Yaskawa INFORM job: N_R2_D7,1(-165,-90)0.JBI

/JOB
//NAME N_R2_D7,1(-165,-90)0
//POS
///NPOS 215,215,215,10,0,0
///TOOL 0
///POSTYPE PULSE
///PULSE
C00000=-39723,-76225,-106677,19950,71807,76871
C00001=-136716,-73683,-105524,19345,72156,77265
C00002=-161407,-91524,-110310,15012,103390,71507
C00003=-134262,-92612,-59078,787,74622,77224
C00004=-134610,-92069,-54626,808,72165,77088
C00005=-134755,-91759,-52790,817,71196,77032
C00006=-134778,-90628,-50545,822,70395,77019
C00007=-134779,-90815,-50888,821,70510,77019
C00008=-134780,-90766,-50877,821,70529,77019
C00009=-135151,-92885,-51740,837,69975,76888
C00010=-134780,-90766,-50877,821,70529,77019
C00011=-134635,-91110,-52736,812,71495,77075
C00012=-134286,-91743,-57244,790,73940,77211
C00013=-131535,-88408,-77632,452,88335,78233
C00014=-134472,-105055,-82285,1702,77673,77142
C00015=-134729,-104914,-78076,1744,75161,77018
C00016=-134834,-104745,-76339,1762,74182,76968
C00017=-134858,-103911,-74317,1771,73367,76948
C00018=-134859,-104062,-74637,1770,73487,76949
C00019=-134909,-103988,-74547,1775,73470,76931
C00020=-135283,-106552,-75509,1819,72754,76790
C00021=-134909,-103988,-74547,1775,73470,76931
C00022=-134803,-104200,-76305,1757,74440,76982
C00023=-134544,-104461,-80571,1713,76925,77107
C00024=-136082,-134381,-102209,6463,55903,75707
C00025=-135108,-114579,-94528,5981,61099,76375
C00026=-134953,-111416,-89269,6014,59485,76347
C00027=-134891,-110125,-87144,6029,58840,76336
C00028=-134915,-109472,-85222,6092,57999,76280
C00029=-134915,-109614,-85578,6083,58144,76288
C00030=-134962,-109452,-85494,6099,58179,76271
C00031=-135337,-112331,-86541,6305,57378,76076
C00032=-134962,-109452,-85494,6099,58179,76271
C00033=-135023,-110765,-87631,6083,58821,76283
C00034=-135179,-113988,-92923,6048,60424,76311
C00035=-156260,-82084,-105549,20460,72443,69801
C00036=-137260,-84248,-120477,10166,77039,76481
C00037=-137260,-138866,-129024,10166,31486,76481
C00038=-31464,-162597,-129024,10166,12061,76481
C00039=11401,-148032,-125424,11666,35639,75770
C00040=126224,-114648,-117374,36487,17100,65054
C00041=160935,-140982,-109639,13467,75088,4607
C00042=171546,-94218,-58921,11830,67408,-77190
C00043=173316,-92720,-54117,11803,65014,-76792
C00044=174042,-92038,-52145,11792,64066,-76624
C00045=174183,-90834,-49869,11851,63281,-76655
C00046=174042,-92038,-52145,11792,64066,-76624
C00047=174177,-91005,-50226,11839,63410,-76643
C00048=175494,-92657,-50922,11711,62814,-76221
C00049=174177,-91005,-50226,11839,63410,-76643
C00050=173449,-91716,-52219,11847,64356,-76811
C00051=171674,-93290,-57074,11869,66744,-77212
C00052=148466,-121612,-87036,17170,72641,-74850
C00053=158367,-105008,-80303,12719,76823,-80933
C00054=159865,-104818,-76175,12706,74203,-80677
C00055=160482,-104628,-74471,12705,73177,-80565
C00056=160593,-103709,-72411,12744,72384,-80610
C00057=160482,-104628,-74471,12705,73177,-80565
C00058=160542,-103788,-72707,12740,72530,-80613
C00059=161564,-106010,-73554,12683,71765,-80329
C00060=160542,-103788,-72707,12740,72530,-80613
C00061=159923,-104017,-74432,12740,73548,-80725
C00062=158422,-104310,-78610,12746,76147,-80984
C00063=158674,-141756,-113025,9949,80411,-74851
C00064=158893,-111477,-96824,9930,85641,-81694
C00065=159967,-112919,-93343,9895,82666,-81559
C00066=160412,-113323,-91879,9887,81519,-81496
C00067=160523,-112689,-89977,9898,80673,-81526
C00068=160509,-112801,-90280,9896,80802,-81520
C00069=160550,-112812,-90284,9894,80794,-81506
C00070=161574,-115499,-91253,9843,79895,-81223
C00071=160550,-112812,-90284,9894,80794,-81506
C00072=160103,-112470,-91772,9900,81925,-81571
C00073=159023,-111201,-95321,9929,84853,-81711
C00074=160752,-88554,-104051,4755,98097,-77411
C00075=135358,-109973,-92009,-1179,81206,-77087
C00076=132931,-92872,-58798,-293,74315,-77659
C00077=133296,-92294,-54326,-308,71862,-77528
C00078=133447,-91972,-52482,-315,70894,-77474
C00079=133488,-90828,-50231,-318,70096,-77458
C00080=133482,-91042,-50637,-317,70236,-77460
C00081=133460,-91107,-50617,-317,70190,-77467
C00082=133801,-93226,-51476,-330,69631,-77349
C00083=133460,-91107,-50617,-317,70190,-77467
C00084=133307,-91465,-52485,-310,71155,-77522
C00085=132941,-92137,-57014,-294,73596,-77654
C00086=138453,-137227,-94273,-1895,68830,-75577
C00087=132988,-105621,-81970,-1125,77172,-77601
C00088=133268,-105409,-77729,-1165,74675,-77481
C00089=133383,-105214,-75980,-1182,73700,-77431
C00090=133423,-104355,-73948,-1190,72892,-77409
C00091=133417,-104520,-74315,-1189,73033,-77413
C00092=133393,-104538,-74287,-1187,73006,-77421
C00093=133734,-107100,-75243,-1226,72284,-77295
C00094=133393,-104538,-74287,-1187,73006,-77421
C00095=133278,-104776,-76057,-1170,73972,-77470
C00096=132997,-105102,-80353,-1129,76444,-77591
C00097=138253,-142244,-101762,-7760,51895,-74453
C00098=133458,-115366,-94293,-4986,60456,-76916
C00099=133364,-112113,-89005,-5028,58873,-76880
C00100=133327,-110790,-86870,-5046,58239,-76865
C00101=133368,-110104,-84936,-5108,57407,-76810
C00102=133362,-110233,-85266,-5098,57543,-76819
C00103=133377,-110217,-85238,-5104,57535,-76813
C00104=133717,-113094,-86276,-5290,56721,-76638
C00105=133377,-110217,-85238,-5104,57535,-76813
C00106=133414,-111565,-87387,-5085,58165,-76828
C00107=133508,-114885,-92709,-5041,59734,-76864
C00108=141804,-106560,-89724,-13944,62113,-73509
C00109=139379,-94179,-83096,-11060,68876,-75147
C00110=139056,-93239,-80222,-11055,67569,-75143
C00111=138655,-90526,-79037,-10882,68167,-75347
C00112=139020,-93447,-81559,-10991,68267,-75222
C00113=135650,-94437,-80689,-10014,66800,-76334
C00114=131133,-95634,-81147,-8583,65949,-77941
C00115=127606,-96266,-81385,-7430,65422,-79216
C00116=127923,-97381,-84321,-7467,66675,-79179
C00117=129037,-107781,-90700,-8626,61514,-78396
C00118=153259,-105355,-101722,-11659,72368,-68227
C00119=139055,-107982,-91136,13627,98522,-80003
C00120=140531,-111621,-88895,13695,95112,-79863
C00121=141160,-112889,-87907,13741,93781,-79791
C00122=141114,-113409,-89355,13751,94395,-79738
C00123=140635,-110012,-86860,13696,94681,-79874
C00124=145054,-111200,-87361,14229,93626,-78446
C00125=149927,-108602,-86499,14790,93534,-76747
C00126=153516,-106318,-85721,15167,93544,-75484
C00127=152717,-105120,-86692,15125,94866,-75603
C00128=150826,-101669,-88898,15064,98245,-75855
C00129=161013,-93310,-79433,24228,97681,-73156
C00130=152044,-102420,-74574,18748,88667,-80737
C00131=154129,-104098,-71555,18965,85609,-80472
C00132=155013,-104629,-70277,19068,84402,-80349
C00133=154938,-105384,-71853,19049,84971,-80287
C00134=154138,-102381,-69420,18973,85198,-80533
C00135=158674,-102440,-69551,19374,84196,-79089
C00136=163166,-99303,-68473,19685,84034,-77522
C00137=166415,-96688,-67542,19865,83984,-76373
C00138=165435,-96203,-68797,19786,85183,-76526
C00139=163100,-94647,-71761,19624,88219,-76868
C00140=177469,-96162,-81466,-5174,90371,-76160
C00141=140989,-97571,-77910,-6477,80304,-75413
C00142=139257,-88771,-70558,-5122,84704,-76235
C00143=139247,-89361,-68393,-5133,83074,-76172
C00144=138839,-86919,-67301,-5121,83628,-76333
C00145=139210,-89792,-69844,-5127,83741,-76212
C00146=135828,-90440,-68818,-5070,82565,-77317
C00147=131175,-91540,-69244,-4968,81974,-78881
C00148=127631,-92103,-69459,-4877,81601,-80076
C00149=127824,-91599,-71673,-4868,83228,-80074
C00150=128905,-101797,-79416,-5532,77763,-79457
C00151=137935,-111344,-72360,-1825,88711,-76983
C00152=138175,-87355,-54576,-1641,89871,-76939
C00153=138462,-88899,-51460,-1591,87166,-76810
C00154=138585,-89409,-50143,-1570,86097,-76756
C00155=138142,-87310,-49251,-1647,86617,-76908
C00156=138544,-90243,-51824,-1577,86701,-76777
C00157=134711,-90264,-50450,-2245,85757,-78018
C00158=129567,-91064,-50732,-3132,85354,-79692
C00159=133440,-90680,-49995,-7180,85761,-79174
C00160=133642,-90171,-51309,-7139,86839,-79169
C00161=134115,-88628,-54418,-7054,89566,-79166
C00162=164381,-109390,-67526,9871,79554,-67793
C00163=178481,-110687,-72352,20846,77564,-61880
C00164=158703,-97120,-53511,19723,77491,-80168
C00165=161312,-97088,-49613,20147,74642,-79736
C00166=162421,-96967,-47993,20332,73505,-79545
C00167=162322,-98010,-49764,20272,74049,-79485
C00168=161267,-95191,-47313,20182,74238,-79821
C00169=166229,-94856,-47327,20585,73246,-78256
C00170=170826,-91864,-46338,20811,73023,-76672
C00171=170725,-92212,-45770,23236,70848,-76635
C00172=169440,-92471,-47412,23069,72000,-76869
C00173=166376,-92848,-51371,22679,74886,-77407
C00174=149893,-144723,-110594,14593,75698,-63607
C00175=126224,-114648,-117374,36487,17100,65054
C00176=118781,-153852,-129024,32591,23356,65054
C00177=12469,-167082,-125424,11666,16324,75770
C00178=-137258,-84249,-120477,10166,64820,76481
C00179=-160540,-100856,-113062,23154,68828,67580
C00180=-142919,-103613,-89511,14221,64514,73447
C00181=-140713,-93202,-83145,11806,69584,74803
C00182=-140366,-92325,-80297,11799,68258,74797
C00183=-140342,-92507,-81623,11736,68962,74877
C00184=-139943,-89620,-79106,11620,68840,75011
C00185=-137000,-93615,-80822,10786,67454,75962
C00186=-132529,-94936,-81358,9390,66550,77539
C00187=-129034,-95667,-81655,8259,65976,78791
C00188=-129377,-96731,-84569,8298,67246,78755
C00189=-130985,-110873,-91431,10312,58832,77470
C00190=-137786,-122665,-93672,6634,76519,76374
C00191=-142705,-98537,-78672,7318,79679,74834
C00192=-140492,-88091,-70749,5581,85268,75891
C00193=-140474,-88727,-68610,5592,83630,75824
C00194=-140449,-89137,-70051,5586,84302,75862
C00195=-140046,-86288,-67512,5580,84176,75994
C00196=-137092,-89887,-69090,5534,83097,76954
C00197=-132483,-91099,-69589,5437,82469,78500
C00198=-128968,-91749,-69858,5349,82066,79683
C00199=-129166,-91202,-72049,5340,83701,79685
C00200=-130908,-106571,-81390,6599,74332,78625
C00201=-147199,-111997,-78117,4842,93237,75003
C00202=-140629,-86347,-53809,6324,90898,77078
C00203=-140437,-88027,-50796,6352,88182,77004
C00204=-140355,-88591,-49520,6369,87107,76977
C00205=-140327,-89422,-51202,6373,87709,77017
C00206=-139876,-86509,-48628,6458,87588,77159
C00207=-136525,-89545,-49887,7080,86535,78207
C00208=-131427,-90479,-50246,8002,85818,79842
C00209=-127439,-90954,-50432,8701,85292,81122
C00210=-127780,-90460,-51749,8636,86380,81084
C00211=-128575,-88953,-54867,8495,89126,81007
C00212=-161407,-91524,-110310,15012,103390,71507
C00213=-136716,-73683,-105524,19345,72156,77265
C00214=-39723,-76225,-106677,19950,71807,76871
BC00000=295325,674563,1075175
BC00001=353535,895977,1075175
BC00002=353535,975867,1075175
BC00003=346138,1016365,1074941
BC00004=346138,1016365,1074941
BC00005=346138,1016365,1074941
BC00006=346138,1016365,1074941
BC00007=346138,1016365,1074941
BC00008=346138,1016365,1074941
BC00009=346138,1016365,1074941
BC00010=346138,1016365,1074941
BC00011=346138,1016365,1074941
BC00012=346138,1016365,1074941
BC00013=345633,1015596,1047596
BC00014=345436,1039539,1075175
BC00015=345436,1039539,1075175
BC00016=345436,1039539,1075175
BC00017=345436,1039539,1075175
BC00018=345436,1039539,1075175
BC00019=345436,1039539,1075175
BC00020=345436,1039539,1075175
BC00021=345436,1039539,1075175
BC00022=345436,1039539,1075175
BC00023=345436,1039539,1075175
BC00024=345633,1030850,1075175
BC00025=346084,1031619,1075175
BC00026=346084,1031619,1075175
BC00027=346084,1031619,1075175
BC00028=346084,1031619,1075175
BC00029=346084,1031619,1075175
BC00030=346084,1031619,1075175
BC00031=346084,1031619,1075175
BC00032=346084,1031619,1075175
BC00033=346084,1031619,1075175
BC00034=346084,1031619,1075175
BC00035=381896,966588,1075175
BC00036=353816,923989,1075175
BC00037=353816,923989,1075175
BC00038=379773,1126391,1075175
BC00039=398190,1030285,1075175
BC00040=312632,1138057,1075175
BC00041=340753,1115300,1075175
BC00042=317618,1085268,1067802
BC00043=317618,1085268,1067802
BC00044=317618,1085268,1067802
BC00045=317618,1085268,1067802
BC00046=317618,1085268,1067802
BC00047=317618,1085268,1067802
BC00048=317618,1085268,1067802
BC00049=317618,1085268,1067802
BC00050=317618,1085268,1067802
BC00051=317618,1085268,1067802
BC00052=304558,1071386,1075175
BC00053=304527,1061353,1075175
BC00054=304527,1061353,1075175
BC00055=304527,1061353,1075175
BC00056=304527,1061353,1075175
BC00057=304527,1061353,1075175
BC00058=304527,1061353,1075175
BC00059=304527,1061353,1075175
BC00060=304527,1061353,1075175
BC00061=304527,1061353,1075175
BC00062=304527,1061353,1075175
BC00063=297809,1030861,1075175
BC00064=297809,1030861,1075175
BC00065=297809,1030861,1075175
BC00066=297809,1030861,1075175
BC00067=297809,1030861,1075175
BC00068=297809,1030861,1075175
BC00069=297809,1030861,1075175
BC00070=297809,1030861,1075175
BC00071=297809,1030861,1075175
BC00072=297809,1030861,1075175
BC00073=297809,1030861,1075175
BC00074=323405,1100688,1075175
BC00075=345633,1145987,1075175
BC00076=345627,1107551,1074273
BC00077=345627,1107551,1074273
BC00078=345627,1107551,1074273
BC00079=345627,1107551,1074273
BC00080=345627,1107551,1074273
BC00081=345627,1107551,1074273
BC00082=345627,1107551,1074273
BC00083=345627,1107551,1074273
BC00084=345627,1107551,1074273
BC00085=345627,1107551,1074273
BC00086=345633,1085057,1075175
BC00087=345596,1084288,1075175
BC00088=345596,1084288,1075175
BC00089=345596,1084288,1075175
BC00090=345596,1084288,1075175
BC00091=345596,1084288,1075175
BC00092=345596,1084288,1075175
BC00093=345596,1084288,1075175
BC00094=345596,1084288,1075175
BC00095=345596,1084288,1075175
BC00096=345596,1084288,1075175
BC00097=345633,1092894,1075175
BC00098=345573,1092125,1075175
BC00099=345573,1092125,1075175
BC00100=345573,1092125,1075175
BC00101=345573,1092125,1075175
BC00102=345573,1092125,1075175
BC00103=345573,1092125,1075175
BC00104=345573,1092125,1075175
BC00105=345573,1092125,1075175
BC00106=345573,1092125,1075175
BC00107=345573,1092125,1075175
BC00108=338421,1101651,1075175
BC00109=338421,1101651,1075175
BC00110=338421,1101651,1075175
BC00111=338421,1101651,1075175
BC00112=338421,1101651,1075175
BC00113=338421,1101651,1075175
BC00114=338421,1101651,1075175
BC00115=338421,1101651,1075175
BC00116=338421,1101651,1075175
BC00117=338421,1101651,1075175
BC00118=329561,1092894,1075175
BC00119=285121,1016140,1075175
BC00120=285121,1016140,1075175
BC00121=285121,1016140,1075175
BC00122=285121,1016140,1075175
BC00123=285121,1016140,1075175
BC00124=285121,1016140,1075175
BC00125=285121,1016140,1075175
BC00126=285121,1016140,1075175
BC00127=285121,1016140,1075175
BC00128=285121,1016140,1075175
BC00129=322883,1030260,1075175
BC00130=305317,1037338,1075175
BC00131=305317,1037338,1075175
BC00132=305317,1037338,1075175
BC00133=305317,1037338,1075175
BC00134=305317,1037338,1075175
BC00135=305317,1037338,1075175
BC00136=305317,1037338,1075175
BC00137=305317,1037338,1075175
BC00138=305317,1037338,1075175
BC00139=305317,1037338,1075175
BC00140=352461,1065435,1075175
BC00141=338520,1089250,1075175
BC00142=338520,1089250,1075175
BC00143=338520,1089250,1075175
BC00144=338520,1089250,1075175
BC00145=338520,1089250,1075175
BC00146=338520,1089250,1075175
BC00147=338520,1089250,1075175
BC00148=338520,1089250,1075175
BC00149=338520,1089250,1075175
BC00150=338520,1089250,1075175
BC00151=329561,1063988,1075175
BC00152=334879,1082600,1057410
BC00153=334879,1082600,1057410
BC00154=334879,1082600,1057410
BC00155=334879,1082600,1057410
BC00156=334879,1082600,1057410
BC00157=334879,1082600,1057410
BC00158=334879,1082600,1057410
BC00159=334879,1082600,1057410
BC00160=334879,1082600,1057410
BC00161=334879,1082600,1057410
BC00162=331300,1058024,1069499
BC00163=329561,1042367,1075175
BC00164=308437,1059196,1075175
BC00165=308437,1059196,1075175
BC00166=308437,1059196,1075175
BC00167=308437,1059196,1075175
BC00168=308437,1059196,1075175
BC00169=308437,1059196,1075175
BC00170=308437,1059196,1075175
BC00171=308437,1059196,1075175
BC00172=308437,1059196,1075175
BC00173=308437,1059196,1075175
BC00174=340753,1115300,1075175
BC00175=312632,1138057,1075175
BC00176=312632,1138057,1075175
BC00177=398190,1030285,1075175
BC00178=353817,923990,1075175
BC00179=381896,966588,1075175
BC00180=338906,1022094,1075175
BC00181=338906,1022094,1075175
BC00182=338906,1022094,1075175
BC00183=338906,1022094,1075175
BC00184=338906,1022094,1075175
BC00185=338906,1022094,1075175
BC00186=338906,1022094,1075175
BC00187=338906,1022094,1075175
BC00188=338906,1022094,1075175
BC00189=338906,1022094,1075175
BC00190=330026,1050278,1075175
BC00191=338884,1034595,1075175
BC00192=338884,1034595,1075175
BC00193=338884,1034595,1075175
BC00194=338884,1034595,1075175
BC00195=338884,1034595,1075175
BC00196=338884,1034595,1075175
BC00197=338884,1034595,1075175
BC00198=338884,1034595,1075175
BC00199=338884,1034595,1075175
BC00200=338884,1034595,1075175
BC00201=330026,1059203,1075175
BC00202=326517,1040873,1058771
BC00203=326517,1040873,1058771
BC00204=326517,1040873,1058771
BC00205=326517,1040873,1058771
BC00206=326517,1040873,1058771
BC00207=326517,1040873,1058771
BC00208=326517,1040873,1058771
BC00209=326517,1040873,1058771
BC00210=326517,1040873,1058771
BC00211=326517,1040873,1058771
BC00212=353535,975867,1075175
BC00213=353535,895977,1075175
BC00214=295325,674563,1075175
EC00000=-1463287,-556475
EC00001=-1463287,-556475
EC00002=-1463287,-556475
EC00003=-1463287,-556475
EC00004=-1463287,-556475
EC00005=-1463287,-556475
EC00006=-1463287,-556475
EC00007=-1463287,-556475
EC00008=-1463287,-556475
EC00009=-1463287,-556475
EC00010=-1463287,-556475
EC00011=-1463287,-556475
EC00012=-1463287,-556475
EC00013=-1463287,-556475
EC00014=-1463287,-556475
EC00015=-1463287,-556475
EC00016=-1463287,-556475
EC00017=-1463287,-556475
EC00018=-1463287,-556475
EC00019=-1463287,-556475
EC00020=-1463287,-556475
EC00021=-1463287,-556475
EC00022=-1463287,-556475
EC00023=-1463287,-556475
EC00024=-1463287,-556475
EC00025=-1463287,-556475
EC00026=-1463287,-556475
EC00027=-1463287,-556475
EC00028=-1463287,-556475
EC00029=-1463287,-556475
EC00030=-1463287,-556475
EC00031=-1463287,-556475
EC00032=-1463287,-556475
EC00033=-1463287,-556475
EC00034=-1463287,-556475
EC00035=-1463287,-556475
EC00036=-1463287,-556475
EC00037=-1463287,-556475
EC00038=-1463287,-556475
EC00039=-1595090,-3837
EC00040=-1729339,556475
EC00041=-1729339,556475
EC00042=-1729339,556475
EC00043=-1729339,556475
EC00044=-1729339,556475
EC00045=-1729339,556475
EC00046=-1729339,556475
EC00047=-1729339,556475
EC00048=-1729339,556475
EC00049=-1729339,556475
EC00050=-1729339,556475
EC00051=-1729339,556475
EC00052=-1729339,556475
EC00053=-1729339,556475
EC00054=-1729339,556475
EC00055=-1729339,556475
EC00056=-1729339,556475
EC00057=-1729339,556475
EC00058=-1729339,556475
EC00059=-1729339,556475
EC00060=-1729339,556475
EC00061=-1729339,556475
EC00062=-1729339,556475
EC00063=-1729339,556475
EC00064=-1729339,556475
EC00065=-1729339,556475
EC00066=-1729339,556475
EC00067=-1729339,556475
EC00068=-1729339,556475
EC00069=-1729339,556475
EC00070=-1729339,556475
EC00071=-1729339,556475
EC00072=-1729339,556475
EC00073=-1729339,556475
EC00074=-1729339,556475
EC00075=-1729339,556475
EC00076=-1729339,556475
EC00077=-1729339,556475
EC00078=-1729339,556475
EC00079=-1729339,556475
EC00080=-1729339,556475
EC00081=-1729339,556475
EC00082=-1729339,556475
EC00083=-1729339,556475
EC00084=-1729339,556475
EC00085=-1729339,556475
EC00086=-1729339,556475
EC00087=-1729339,556475
EC00088=-1729339,556475
EC00089=-1729339,556475
EC00090=-1729339,556475
EC00091=-1729339,556475
EC00092=-1729339,556475
EC00093=-1729339,556475
EC00094=-1729339,556475
EC00095=-1729339,556475
EC00096=-1729339,556475
EC00097=-1729339,556475
EC00098=-1729339,556475
EC00099=-1729339,556475
EC00100=-1729339,556475
EC00101=-1729339,556475
EC00102=-1729339,556475
EC00103=-1729339,556475
EC00104=-1729339,556475
EC00105=-1729339,556475
EC00106=-1729339,556475
EC00107=-1729339,556475
EC00108=-1729339,556475
EC00109=-1729339,556475
EC00110=-1729339,556475
EC00111=-1729339,556475
EC00112=-1729339,556475
EC00113=-1729339,556475
EC00114=-1729339,556475
EC00115=-1729339,556475
EC00116=-1729339,556475
EC00117=-1729339,556475
EC00118=-1729339,556475
EC00119=-1729339,556475
EC00120=-1729339,556475
EC00121=-1729339,556475
EC00122=-1729339,556475
EC00123=-1729339,556475
EC00124=-1729339,556475
EC00125=-1729339,556475
EC00126=-1729339,556475
EC00127=-1729339,556475
EC00128=-1729339,556475
EC00129=-1729339,556475
EC00130=-1729339,556475
EC00131=-1729339,556475
EC00132=-1729339,556475
EC00133=-1729339,556475
EC00134=-1729339,556475
EC00135=-1729339,556475
EC00136=-1729339,556475
EC00137=-1729339,556475
EC00138=-1729339,556475
EC00139=-1729339,556475
EC00140=-1729339,556475
EC00141=-1729339,556475
EC00142=-1729339,556475
EC00143=-1729339,556475
EC00144=-1729339,556475
EC00145=-1729339,556475
EC00146=-1729339,556475
EC00147=-1729339,556475
EC00148=-1729339,556475
EC00149=-1729339,556475
EC00150=-1729339,556475
EC00151=-1729339,556475
EC00152=-1729339,556475
EC00153=-1729339,556475
EC00154=-1729339,556475
EC00155=-1729339,556475
EC00156=-1729339,556475
EC00157=-1729339,556475
EC00158=-1729339,556475
EC00159=-1729339,556475
EC00160=-1729339,556475
EC00161=-1729339,556475
EC00162=-1729339,556475
EC00163=-1729339,556475
EC00164=-1729339,556475
EC00165=-1729339,556475
EC00166=-1729339,556475
EC00167=-1729339,556475
EC00168=-1729339,556475
EC00169=-1729339,556475
EC00170=-1729339,556475
EC00171=-1729339,556475
EC00172=-1729339,556475
EC00173=-1729339,556475
EC00174=-1729339,556475
EC00175=-1729339,556475
EC00176=-1729339,556475
EC00177=-1595090,-3837
EC00178=-1463287,-556475
EC00179=-1463287,-556475
EC00180=-1463287,-556475
EC00181=-1463287,-556475
EC00182=-1463287,-556475
EC00183=-1463287,-556475
EC00184=-1463287,-556475
EC00185=-1463287,-556475
EC00186=-1463287,-556475
EC00187=-1463287,-556475
EC00188=-1463287,-556475
EC00189=-1463287,-556475
EC00190=-1463287,-556475
EC00191=-1463287,-556475
EC00192=-1463287,-556475
EC00193=-1463287,-556475
EC00194=-1463287,-556475
EC00195=-1463287,-556475
EC00196=-1463287,-556475
EC00197=-1463287,-556475
EC00198=-1463287,-556475
EC00199=-1463287,-556475
EC00200=-1463287,-556475
EC00201=-1463287,-556475
EC00202=-1463287,-556475
EC00203=-1463287,-556475
EC00204=-1463287,-556475
EC00205=-1463287,-556475
EC00206=-1463287,-556475
EC00207=-1463287,-556475
EC00208=-1463287,-556475
EC00209=-1463287,-556475
EC00210=-1463287,-556475
EC00211=-1463287,-556475
EC00212=-1463287,-556475
EC00213=-1463287,-556475
EC00214=-1463287,-556475
///POSTYPE BASE
///RECTAN
///RCONF 0,0,0,0,0,0,0,0,0,0,0,0,0,0,0,0,0,0,0,0,0,0,0,0
P00006=0.222,-3.123,-1.508,0.0000,0.0000,0.0000
P00021=-0.225,-6.128,-0.405,0.0000,0.0000,0.0000
P00022=0.222,-3.123,-1.508,0.0000,0.0000,0.0000
P00023=0.143,-0.036,0.682,0.0000,0.0000,0.0000
P00031=1.853,-0.001,-1.549,0.0000,0.0000,0.0000
P00032=1.957,0.503,-7.217,0.0000,0.0000,0.0000
///RCONF 0,0,0,0,1,0,0,0,0,0,0,0,0,0,0,0,0,0,0,0,0,0,0,0
P00033=-0.123,0.612,-5.012,0.0000,0.0000,0.0000
///RCONF 0,0,0,0,0,0,0,0,0,0,0,0,0,0,0,0,0,0,0,0,0,0,0,0
P00034=-0.304,0.773,-2.693,0.0000,0.0000,0.0000
P00035=2.817,0.591,-1.622,0.0000,0.0000,0.0000
P00036=-1.108,-0.829,1.850,0.0000,0.0000,0.0000
//INST
///DATE 2024/02/02 10:16
///ATTR SC,RW
///GROUP1 RB1,BS1
///GROUP2 ST1
NOP
'N_r2_D7,1(-165,-90)0
MOVJ C00000 BC00000 VJ=100.00  +MOVJ EC00000 VJ=100.00
CALL JOB:CLEAN-R1
MOVJ C00001 BC00001 VJ=100.00  +MOVJ EC00001 VJ=100.00
MOVJ C00002 BC00002 VJ=100.00  +MOVJ EC00002 VJ=100.00
'Path S3195
SSFTOF
MOVJ C00003 BC00003 VJ=100.00  +MOVJ EC00003 VJ=100.00
MOVL C00004 BC00004 V=400.0  +MOVJ EC00004 VJ=100.00
SMOVL C00005 BC00005 V=60.0  +MOVJ EC00005
SREFP 3 C00006 BC00006  +REFP EC00006
CALL JOB:SEARCH-R1-S1
SET P021 P006
SSFTON P021
SMOVL C00007 BC00007 V=60.0  +MOVJ EC00007
SMOVL C00008 BC00008 V=60.0  +MOVJ EC00008
SREFP 3 C00009 BC00009  +REFP EC00009
CALL JOB:SEARCH-R1-S1
SET P021 P006
SSFTON P021
SMOVL C00010 BC00010 V=60.0  +MOVJ EC00010
MOVL C00011 BC00011 V=400.0  +MOVJ EC00011 VJ=100.00
MOVL C00012 BC00012 V=1000.0  +MOVJ EC00012 VJ=100.00
MOVJ C00013 BC00013 VJ=100.00  +MOVJ EC00013 VJ=100.00
'Path S3196
SSFTOF
MOVJ C00014 BC00014 VJ=100.00  +MOVJ EC00014 VJ=100.00
MOVL C00015 BC00015 V=400.0  +MOVJ EC00015 VJ=100.00
SMOVL C00016 BC00016 V=60.0  +MOVJ EC00016
SREFP 3 C00017 BC00017  +REFP EC00017
CALL JOB:SEARCH-R1-S1
SET P022 P006
SSFTON P022
SMOVL C00018 BC00018 V=60.0  +MOVJ EC00018
SMOVL C00019 BC00019 V=60.0  +MOVJ EC00019
SREFP 3 C00020 BC00020  +REFP EC00020
CALL JOB:SEARCH-R1-S1
SET P022 P006
SSFTON P022
SMOVL C00021 BC00021 V=60.0  +MOVJ EC00021
MOVL C00022 BC00022 V=400.0  +MOVJ EC00022 VJ=100.00
MOVL C00023 BC00023 V=1000.0  +MOVJ EC00023 VJ=100.00
MOVJ C00024 BC00024 VJ=100.00  +MOVJ EC00024 VJ=100.00
'Path S3197
SSFTOF
MOVJ C00025 BC00025 VJ=100.00  +MOVJ EC00025 VJ=100.00
MOVL C00026 BC00026 V=400.0  +MOVJ EC00026 VJ=100.00
SMOVL C00027 BC00027 V=60.0  +MOVJ EC00027
SREFP 3 C00028 BC00028  +REFP EC00028
CALL JOB:SEARCH-R1-S1
SET P023 P006
SSFTON P023
SMOVL C00029 BC00029 V=60.0  +MOVJ EC00029
SMOVL C00030 BC00030 V=60.0  +MOVJ EC00030
SREFP 3 C00031 BC00031  +REFP EC00031
CALL JOB:SEARCH-R1-S1
SET P023 P006
SSFTON P023
SMOVL C00032 BC00032 V=60.0  +MOVJ EC00032
MOVL C00033 BC00033 V=400.0  +MOVJ EC00033 VJ=100.00
MOVL C00034 BC00034 V=1000.0  +MOVJ EC00034 VJ=100.00
'obrot
MOVJ C00035 BC00035 VJ=100.00  +MOVJ EC00035 VJ=100.00
MOVJ C00036 BC00036 VJ=100.00  +MOVJ EC00036 VJ=100.00
MOVJ C00037 BC00037 VJ=100.00  +MOVJ EC00037 VJ=100.00
MOVJ C00038 BC00038 VJ=100.00  +MOVJ EC00038 VJ=100.00
MOVJ C00039 BC00039 VJ=100.00  +MOVJ EC00039 VJ=100.00
MOVJ C00040 BC00040 VJ=100.00  +MOVJ EC00040 VJ=100.00
MOVJ C00041 BC00041 VJ=100.00  +MOVJ EC00041 VJ=100.00
'
'Path S3198
SSFTOF
MOVJ C00042 BC00042 VJ=100.00  +MOVJ EC00042 VJ=100.00
MOVL C00043 BC00043 V=400.0  +MOVJ EC00043 VJ=100.00
SMOVL C00044 BC00044 V=60.0  +MOVJ EC00044
SREFP 3 C00045 BC00045  +REFP EC00045
CALL JOB:SEARCH-R1-S1
SET P031 P006
SSFTON P031
SMOVL C00046 BC00046 V=60.0  +MOVJ EC00046
SMOVL C00047 BC00047 V=60.0  +MOVJ EC00047
SREFP 3 C00048 BC00048  +REFP EC00048
CALL JOB:SEARCH-R1-S1
SET P031 P006
SSFTON P031
SMOVL C00049 BC00049 V=60.0  +MOVJ EC00049
MOVL C00050 BC00050 V=400.0  +MOVJ EC00050 VJ=100.00
MOVL C00051 BC00051 V=1000.0  +MOVJ EC00051 VJ=100.00
MOVJ C00052 BC00052 VJ=100.00  +MOVJ EC00052 VJ=100.00
'Path S3199
SSFTOF
MOVJ C00053 BC00053 VJ=100.00  +MOVJ EC00053 VJ=100.00
MOVL C00054 BC00054 V=400.0  +MOVJ EC00054 VJ=100.00
SMOVL C00055 BC00055 V=60.0  +MOVJ EC00055
SREFP 3 C00056 BC00056  +REFP EC00056
CALL JOB:SEARCH-R1-S1
SET P032 P006
SSFTON P032
SMOVL C00057 BC00057 V=60.0  +MOVJ EC00057
SMOVL C00058 BC00058 V=60.0  +MOVJ EC00058
SREFP 3 C00059 BC00059  +REFP EC00059
CALL JOB:SEARCH-R1-S1
SET P032 P006
SSFTON P032
SMOVL C00060 BC00060 V=60.0  +MOVJ EC00060
MOVL C00061 BC00061 V=400.0  +MOVJ EC00061 VJ=100.00
MOVL C00062 BC00062 V=1000.0  +MOVJ EC00062 VJ=100.00
MOVJ C00063 BC00063 VJ=100.00  +MOVJ EC00063 VJ=100.00
'Path S3200
SSFTOF
MOVJ C00064 BC00064 VJ=100.00  +MOVJ EC00064 VJ=100.00
MOVL C00065 BC00065 V=400.0  +MOVJ EC00065 VJ=100.00
SMOVL C00066 BC00066 V=60.0  +MOVJ EC00066
SREFP 3 C00067 BC00067  +REFP EC00067
CALL JOB:SEARCH-R1-S1
SET P033 P006
SSFTON P033
SMOVL C00068 BC00068 V=60.0  +MOVJ EC00068
SMOVL C00069 BC00069 V=60.0  +MOVJ EC00069
SREFP 3 C00070 BC00070  +REFP EC00070
CALL JOB:SEARCH-R1-S1
SET P033 P006
SSFTON P033
SMOVL C00071 BC00071 V=60.0  +MOVJ EC00071
MOVL C00072 BC00072 V=400.0  +MOVJ EC00072 VJ=100.00
MOVL C00073 BC00073 V=1000.0  +MOVJ EC00073 VJ=100.00
MOVJ C00074 BC00074 VJ=100.00  +MOVJ EC00074 VJ=100.00
MOVJ C00075 BC00075 VJ=100.00  +MOVJ EC00075 VJ=100.00
'Path S3201
SSFTOF
MOVJ C00076 BC00076 VJ=100.00  +MOVJ EC00076 VJ=100.00
MOVL C00077 BC00077 V=400.0  +MOVJ EC00077 VJ=100.00
SMOVL C00078 BC00078 V=60.0  +MOVJ EC00078
SREFP 3 C00079 BC00079  +REFP EC00079
CALL JOB:SEARCH-R1-S1
SET P034 P006
SSFTON P034
SMOVL C00080 BC00080 V=60.0  +MOVJ EC00080
SMOVL C00081 BC00081 V=60.0  +MOVJ EC00081
SREFP 3 C00082 BC00082  +REFP EC00082
CALL JOB:SEARCH-R1-S1
SET P034 P006
SSFTON P034
SMOVL C00083 BC00083 V=60.0  +MOVJ EC00083
MOVL C00084 BC00084 V=400.0  +MOVJ EC00084 VJ=100.00
MOVL C00085 BC00085 V=1000.0  +MOVJ EC00085 VJ=100.00
MOVJ C00086 BC00086 VJ=100.00  +MOVJ EC00086 VJ=100.00
'Path S3202
SSFTOF
MOVJ C00087 BC00087 VJ=100.00  +MOVJ EC00087 VJ=100.00
MOVL C00088 BC00088 V=400.0  +MOVJ EC00088 VJ=100.00
SMOVL C00089 BC00089 V=60.0  +MOVJ EC00089
SREFP 3 C00090 BC00090  +REFP EC00090
CALL JOB:SEARCH-R1-S1
SET P035 P006
SSFTON P035
SMOVL C00091 BC00091 V=60.0  +MOVJ EC00091
SMOVL C00092 BC00092 V=60.0  +MOVJ EC00092
SREFP 3 C00093 BC00093  +REFP EC00093
CALL JOB:SEARCH-R1-S1
SET P035 P006
SSFTON P035
SMOVL C00094 BC00094 V=60.0  +MOVJ EC00094
MOVL C00095 BC00095 V=400.0  +MOVJ EC00095 VJ=100.00
MOVL C00096 BC00096 V=1000.0  +MOVJ EC00096 VJ=100.00
MOVJ C00097 BC00097 VJ=100.00  +MOVJ EC00097 VJ=100.00
'Path S3203
SSFTOF
MOVJ C00098 BC00098 VJ=100.00  +MOVJ EC00098 VJ=100.00
MOVL C00099 BC00099 V=400.0  +MOVJ EC00099 VJ=100.00
SMOVL C00100 BC00100 V=60.0  +MOVJ EC00100
SREFP 3 C00101 BC00101  +REFP EC00101
CALL JOB:SEARCH-R1-S1
SET P036 P006
SSFTON P036
SMOVL C00102 BC00102 V=60.0  +MOVJ EC00102
SMOVL C00103 BC00103 V=60.0  +MOVJ EC00103
SREFP 3 C00104 BC00104  +REFP EC00104
CALL JOB:SEARCH-R1-S1
SET P036 P006
SSFTON P036
SMOVL C00105 BC00105 V=60.0  +MOVJ EC00105
MOVL C00106 BC00106 V=400.0  +MOVJ EC00106 VJ=100.00
MOVL C00107 BC00107 V=1000.0  +MOVJ EC00107 VJ=100.00
'Path W3204
SSFTOF
SSFTON P036
MOVJ C00108 BC00108 VJ=100.00  +MOVJ EC00108 VJ=100.00
SMOVL C00109 BC00109 V=400.0  +MOVJ EC00109
SMOVL C00110 BC00110 V=100.0 PL=0  +MOVJ EC00110
SREFP 1 C00111 BC00111  +REFP EC00111
SREFP 2 C00112 BC00112  +REFP EC00112
MACRO1 MJ#(0) ARGF0
ARCON
SMOVL C00113 BC00113 V=10.0  +MOVJ EC00113
SMOVL C00114 BC00114 V=10.0  +MOVJ EC00114
SMOVL C00115 BC00115 V=10.0  +MOVJ EC00115
ARCOF
SMOVL C00116 BC00116 V=400.0  +MOVJ EC00116
SMOVL C00117 BC00117 V=1000.0  +MOVJ EC00117
SSFTOF
MOVJ C00118 BC00118 VJ=100.00  +MOVJ EC00118 VJ=100.00
'Path W3205
SSFTOF
SSFTON P033
MOVJ C00119 BC00119 VJ=100.00  +MOVJ EC00119 VJ=100.00
SMOVL C00120 BC00120 V=400.0  +MOVJ EC00120
SMOVL C00121 BC00121 V=100.0 PL=0  +MOVJ EC00121
SREFP 1 C00122 BC00122  +REFP EC00122
SREFP 2 C00123 BC00123  +REFP EC00123
MACRO1 MJ#(0) ARGF0
ARCON
SMOVL C00124 BC00124 V=10.0  +MOVJ EC00124
SMOVL C00125 BC00125 V=10.0  +MOVJ EC00125
SMOVL C00126 BC00126 V=10.0  +MOVJ EC00126
ARCOF
SMOVL C00127 BC00127 V=400.0  +MOVJ EC00127
SMOVL C00128 BC00128 V=1000.0  +MOVJ EC00128
SSFTOF
MOVJ C00129 BC00129 VJ=100.00  +MOVJ EC00129 VJ=100.00
'Path W3206
SSFTOF
SSFTON P032
MOVJ C00130 BC00130 VJ=100.00  +MOVJ EC00130 VJ=100.00
SMOVL C00131 BC00131 V=400.0  +MOVJ EC00131
SMOVL C00132 BC00132 V=100.0 PL=0  +MOVJ EC00132
SREFP 1 C00133 BC00133  +REFP EC00133
SREFP 2 C00134 BC00134  +REFP EC00134
MACRO1 MJ#(0) ARGF0
ARCON
SMOVL C00135 BC00135 V=10.0  +MOVJ EC00135
SMOVL C00136 BC00136 V=10.0  +MOVJ EC00136
SMOVL C00137 BC00137 V=10.0  +MOVJ EC00137
ARCOF
SMOVL C00138 BC00138 V=400.0  +MOVJ EC00138
SMOVL C00139 BC00139 V=1000.0  +MOVJ EC00139
SSFTOF
MOVJ C00140 BC00140 VJ=100.00  +MOVJ EC00140 VJ=100.00
'Path W3207
SSFTOF
SSFTON P035
MOVJ C00141 BC00141 VJ=100.00  +MOVJ EC00141 VJ=100.00
SMOVL C00142 BC00142 V=400.0  +MOVJ EC00142
SMOVL C00143 BC00143 V=100.0 PL=0  +MOVJ EC00143
SREFP 1 C00144 BC00144  +REFP EC00144
SREFP 2 C00145 BC00145  +REFP EC00145
MACRO1 MJ#(0) ARGF0
ARCON
SMOVL C00146 BC00146 V=10.0  +MOVJ EC00146
SMOVL C00147 BC00147 V=10.0  +MOVJ EC00147
SMOVL C00148 BC00148 V=10.0  +MOVJ EC00148
ARCOF
SMOVL C00149 BC00149 V=400.0  +MOVJ EC00149
SMOVL C00150 BC00150 V=1000.0  +MOVJ EC00150
SSFTOF
MOVJ C00151 BC00151 VJ=100.00  +MOVJ EC00151 VJ=100.00
'Path W3208
SSFTOF
SSFTON P034
MOVJ C00152 BC00152 VJ=100.00  +MOVJ EC00152 VJ=100.00
SMOVL C00153 BC00153 V=400.0  +MOVJ EC00153
SMOVL C00154 BC00154 V=100.0 PL=0  +MOVJ EC00154
SREFP 1 C00155 BC00155  +REFP EC00155
SREFP 2 C00156 BC00156  +REFP EC00156
MACRO1 MJ#(0) ARGF0
ARCON
SMOVL C00157 BC00157 V=10.0  +MOVJ EC00157
SMOVL C00158 BC00158 V=10.0  +MOVJ EC00158
SMOVL C00159 BC00159 V=10.0  +MOVJ EC00159
ARCOF
SMOVL C00160 BC00160 V=400.0  +MOVJ EC00160
SMOVL C00161 BC00161 V=1000.0  +MOVJ EC00161
SSFTOF
MOVJ C00162 BC00162 VJ=100.00  +MOVJ EC00162 VJ=100.00
MOVJ C00163 BC00163 VJ=100.00  +MOVJ EC00163 VJ=100.00
'Path W3209
SSFTOF
SSFTON P031
MOVJ C00164 BC00164 VJ=100.00  +MOVJ EC00164 VJ=100.00
SMOVL C00165 BC00165 V=400.0  +MOVJ EC00165
SMOVL C00166 BC00166 V=100.0 PL=0  +MOVJ EC00166
SREFP 1 C00167 BC00167  +REFP EC00167
SREFP 2 C00168 BC00168  +REFP EC00168
MACRO1 MJ#(0) ARGF0
ARCON
SMOVL C00169 BC00169 V=10.0  +MOVJ EC00169
SMOVL C00170 BC00170 V=10.0  +MOVJ EC00170
SMOVL C00171 BC00171 V=10.0  +MOVJ EC00171
ARCOF
SMOVL C00172 BC00172 V=400.0  +MOVJ EC00172
SMOVL C00173 BC00173 V=1000.0  +MOVJ EC00173
SSFTOF
'obrot
MOVJ C00174 BC00174 VJ=100.00  +MOVJ EC00174 VJ=100.00
MOVJ C00175 BC00175 VJ=100.00  +MOVJ EC00175 VJ=100.00
MOVJ C00176 BC00176 VJ=100.00  +MOVJ EC00176 VJ=100.00
MOVJ C00177 BC00177 VJ=100.00  +MOVJ EC00177 VJ=100.00
MOVJ C00178 BC00178 VJ=100.00  +MOVJ EC00178 VJ=100.00
MOVJ C00179 BC00179 VJ=100.00  +MOVJ EC00179 VJ=100.00
'
'Path W3210
SSFTOF
SSFTON P023
MOVJ C00180 BC00180 VJ=100.00  +MOVJ EC00180 VJ=100.00
SMOVL C00181 BC00181 V=400.0  +MOVJ EC00181
SMOVL C00182 BC00182 V=100.0 PL=0  +MOVJ EC00182
SREFP 1 C00183 BC00183  +REFP EC00183
SREFP 2 C00184 BC00184  +REFP EC00184
MACRO1 MJ#(0) ARGF0
ARCON
SMOVL C00185 BC00185 V=10.0  +MOVJ EC00185
SMOVL C00186 BC00186 V=10.0  +MOVJ EC00186
SMOVL C00187 BC00187 V=10.0  +MOVJ EC00187
ARCOF
SMOVL C00188 BC00188 V=400.0  +MOVJ EC00188
SMOVL C00189 BC00189 V=1000.0  +MOVJ EC00189
SSFTOF
MOVJ C00190 BC00190 VJ=100.00  +MOVJ EC00190 VJ=100.00
'Path W3211
SSFTOF
SSFTON P022
MOVJ C00191 BC00191 VJ=100.00  +MOVJ EC00191 VJ=100.00
SMOVL C00192 BC00192 V=400.0  +MOVJ EC00192
SMOVL C00193 BC00193 V=100.0 PL=0  +MOVJ EC00193
SREFP 1 C00194 BC00194  +REFP EC00194
SREFP 2 C00195 BC00195  +REFP EC00195
MACRO1 MJ#(0) ARGF0
ARCON
SMOVL C00196 BC00196 V=10.0  +MOVJ EC00196
SMOVL C00197 BC00197 V=10.0  +MOVJ EC00197
SMOVL C00198 BC00198 V=10.0  +MOVJ EC00198
ARCOF
SMOVL C00199 BC00199 V=400.0  +MOVJ EC00199
SMOVL C00200 BC00200 V=1000.0  +MOVJ EC00200
SSFTOF
MOVJ C00201 BC00201 VJ=100.00  +MOVJ EC00201 VJ=100.00
'Path W3212
SSFTOF
SSFTON P021
MOVJ C00202 BC00202 VJ=100.00  +MOVJ EC00202 VJ=100.00
SMOVL C00203 BC00203 V=400.0  +MOVJ EC00203
SMOVL C00204 BC00204 V=100.0 PL=0  +MOVJ EC00204
SREFP 1 C00205 BC00205  +REFP EC00205
SREFP 2 C00206 BC00206  +REFP EC00206
MACRO1 MJ#(0) ARGF0
ARCON
SMOVL C00207 BC00207 V=10.0  +MOVJ EC00207
SMOVL C00208 BC00208 V=10.0  +MOVJ EC00208
SMOVL C00209 BC00209 V=10.0  +MOVJ EC00209
ARCOF
SMOVL C00210 BC00210 V=400.0  +MOVJ EC00210
SMOVL C00211 BC00211 V=1000.0  +MOVJ EC00211
SSFTOF
MOVJ C00212 BC00212 VJ=100.00  +MOVJ EC00212 VJ=100.00
MOVJ C00213 BC00213 VJ=100.00  +MOVJ EC00213 VJ=100.00
MOVJ C00214 BC00214 VJ=100.00  +MOVJ EC00214 VJ=100.00
END
